// TIA Portal V19 export
TYPE "LEXCHANGETRAY_typeEmActionManager"
// stored: Access Published
   STRUCT
      init : Bool;
      actionEMConstraint : "LEXCHANGETRAY_typeEmActionCostraint";
      actionEMPlastic { S7_SetPoint := 'True'} : "LEXCHANGETRAY_typeEmActionPlastic";
   END_STRUCT;
END_TYPE
